FUNCTION FC_myDTtoString : STRING
VAR_INPUT
	in		: STRING;

END_VAR
VAR
	tempString : ARRAY[0..2] OF STRING;
	pos : INT;
END_VAR

tempString[0] := DELETE(in, 3, 1);
pos := FIND(tempString[0], '-');
tempString[1] := tempString[0];
WHILE pos > 0 DO
	tempString[1] := REPLACE(tempString[1], '_', 1, pos);
	pos := FIND(tempString[1], '-');
END_WHILE

pos := FIND(tempString[1], ':');
tempString[2] := tempString[1];
WHILE pos > 0 DO
	tempString[2] := REPLACE(tempString[2], '_', 1, pos);
	pos := FIND(tempString[2], ':');
END_WHILE

FC_myDTtoString := tempString[2];

END_FUNCTION

(* stored: Version 1.1.0.1, ProductVersion 3.1.4024.15
   POU FC_myDTtoString: Id {9bdc73a8-4fb8-4117-b0a1-56ad98b0f462}, SpecialFunc None *)
